FUNCTION RFID_Sensor_Wread : BOOL
VAR_INPUT
	Data : REFERENCE TO RFID_Tag_Data;
	P : UINT;
END_VAR
VAR_IN_OUT
	Sensor : RFID_Sensor;
END_VAR

IF (P < 64) AND (Sensor.State = RFID_SensorState.idel) THEN
	Sensor.State := RFID_SensorState.WreadTag;
	Sensor.WreadState := Wread_State.Triggerd;
	Sensor.Pagina := P;
	Sensor.TxBuffer := Data.Data;
END_IF

END_FUNCTION

(* stored: Version 1.1.0.1, ProductVersion 3.1.4024.10
   POU RFID_Sensor_Wread: Id {6df75545-5aac-4941-aef3-b7dd09fa2706}, SpecialFunc None *)
